% RSLogix 500 project EDINBURG.RSS, saved by version 10.00.00.00 %
PROJECT "EDINBURG"    % processor: MicroLogix 1400 %

PROGRAM FILES
  LAD 2 "MAIN"  12 rungs
  LAD 3 "START/MODE"  11 rungs
  LAD 4 "ENCODER"  11 rungs
  LAD 5 "CRADLE"  25 rungs
  LAD 6 "BRUSH"  8 rungs
  LAD 7 "TANK"  17 rungs
  LAD 8 "AUXILARY"  4 rungs
  LAD 9 "FAULTS"  35 rungs
  LAD 10 "SPARE"  2 rungs
  LAD 11 "DECLINE"  49 rungs
  LAD 12 "STACK LS"  13 rungs
  LAD 13 "STACK"  23 rungs

DATA FILES
  O0 OUTPUT  9 elements
  I1 INPUT  11 elements
  S2 STATUS  66 elements
  B3 BINARY  7 elements
  T4 TIMER  38 elements
  C5 COUNTER  1 elements
  R6 CONTROL  1 elements
  N7 INTEGER  40 elements
  F8 FLOAT  30 elements
  L9   1 elements
  L10   2 elements

LADDER 2 "MAIN"
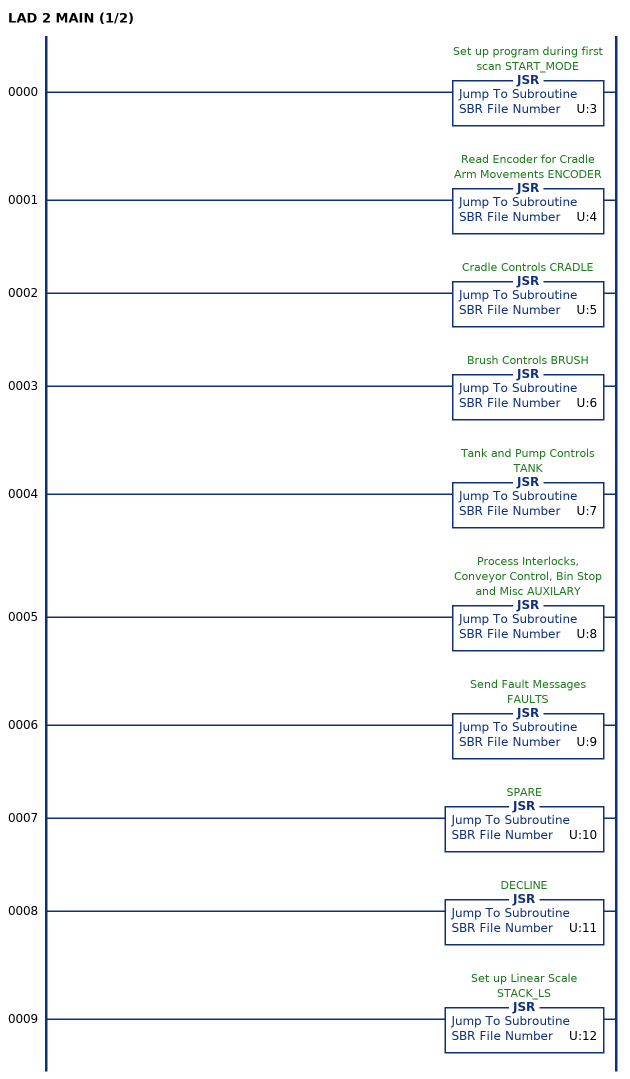
% Rung: 0 %
SOR JSR U:3 EOR
%   U:3  START_MODE  "Set up program during first scan" %
% Rung: 1 %
SOR JSR U:4 EOR
%   U:4  ENCODER  "Read Encoder for Cradle Arm Movements" %
% Rung: 2 %
SOR JSR U:5 EOR
%   U:5  CRADLE  "Cradle Controls" %
% Rung: 3 %
SOR JSR U:6 EOR
%   U:6  BRUSH  "Brush Controls" %
% Rung: 4 %
SOR JSR U:7 EOR
%   U:7  TANK  "Tank and Pump Controls" %
% Rung: 5 %
SOR JSR U:8 EOR
%   U:8  AUXILARY  "Process Interlocks, Conveyor Control, Bin Stop and Misc" %
% Rung: 6 %
SOR JSR U:9 EOR
%   U:9  FAULTS  "Send Fault Messages" %
% Rung: 7 %
SOR JSR U:10 EOR
%   U:10  SPARE %
% Rung: 8 %
SOR JSR U:11 EOR
%   U:11  DECLINE %
% Rung: 9 %
SOR JSR U:12 EOR
%   U:12  STACK_LS  "Set up Linear Scale" %

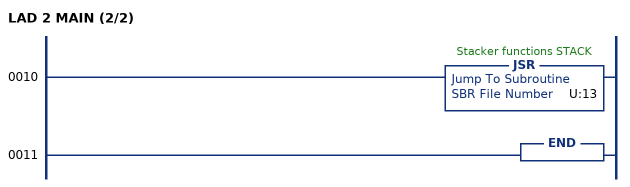
% Rung: 10 %
SOR JSR U:13 EOR
%   U:13  STACK  "Stacker functions" %
% Rung: 11 %
SOR END EOR

LADDER 3 "START/MODE"
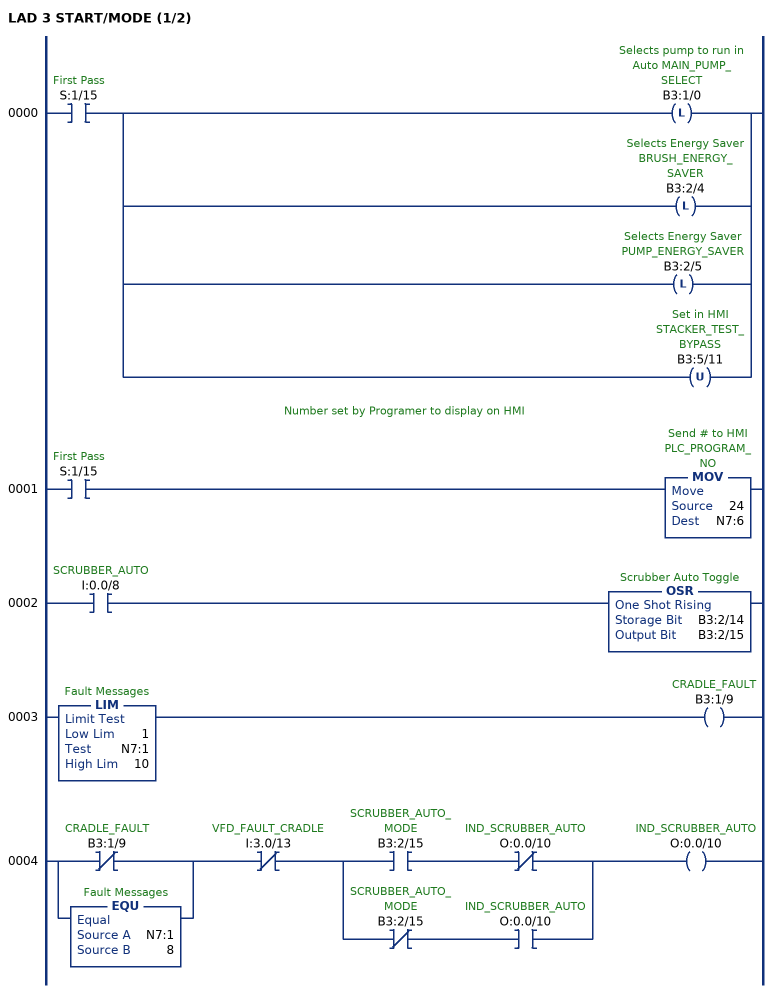
% Rung: 0 %
SOR XIC S:1/15 BST OTL B3:1/0 NXB BST OTL B3:2/4 NXB BST OTL B3:2/5 NXB OTU B3:5/11 BND BND BND EOR
%   S:1/15  "First Pass" %
%   B3:1/0  MAIN_PUMP_SELECT  "Selects pump to run in Auto" %
%   B3:2/4  BRUSH_ENERGY_SAVER  "Selects Energy Saver" %
%   B3:2/5  PUMP_ENERGY_SAVER  "Selects Energy Saver" %
%   B3:5/11  STACKER_TEST_BYPASS  "Set in HMI" %
% Rung: 1 %
% Number set by Programer to display on HMI %
SOR XIC S:1/15 MOV 24 N7:6 EOR
%   S:1/15  "First Pass" %
%   N7:6  PLC_PROGRAM_NO  "Send # to HMI" %
% Rung: 2 %
SOR XIC I:0.0/8 OSR B3:2/14 B3:2/15 EOR
%   I:0.0/8  SCRUBBER_AUTO %
%   B3:2/14  "Scrubber Auto Toggle" %
%   B3:2/15  SCRUBBER_AUTO_MODE %
% Rung: 3 %
SOR LIM 1 N7:1 10 OTE B3:1/9 EOR
%   N7:1  "Fault Messages" %
%   B3:1/9  CRADLE_FAULT %
% Rung: 4 %
SOR BST XIO B3:1/9 NXB EQU N7:1 8 BND XIO I:3.0/13 BST XIC B3:2/15 XIO O:0.0/10 NXB XIO B3:2/15 XIC O:0.0/10 BND OTE O:0.0/10 EOR
%   B3:1/9  CRADLE_FAULT %
%   N7:1  "Fault Messages" %
%   I:3.0/13  VFD_FAULT_CRADLE %
%   B3:2/15  SCRUBBER_AUTO_MODE %
%   O:0.0/10  IND_SCRUBBER_AUTO %

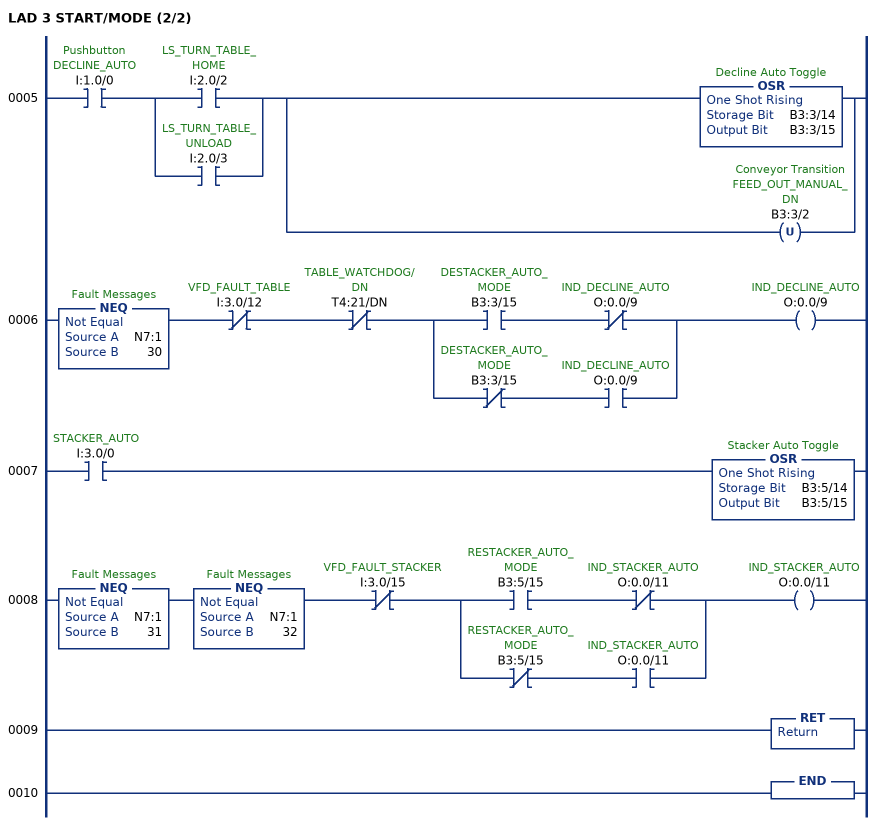
% Rung: 5 %
SOR XIC I:1.0/0 BST XIC I:2.0/2 NXB XIC I:2.0/3 BND BST OSR B3:3/14 B3:3/15 NXB OTU B3:3/2 BND EOR
%   I:1.0/0  DECLINE_AUTO  "Pushbutton" %
%   I:2.0/2  LS_TURN_TABLE_HOME %
%   I:2.0/3  LS_TURN_TABLE_UNLOAD %
%   B3:3/14  "Decline Auto Toggle" %
%   B3:3/15  DESTACKER_AUTO_MODE %
%   B3:3/2  FEED_OUT_MANUAL_DN  "Conveyor Transition" %
% Rung: 6 %
SOR NEQ N7:1 30 XIO I:3.0/12 XIO T4:21/DN BST XIC B3:3/15 XIO O:0.0/9 NXB XIO B3:3/15 XIC O:0.0/9 BND OTE O:0.0/9 EOR
%   N7:1  "Fault Messages" %
%   I:3.0/12  VFD_FAULT_TABLE %
%   T4:21  TABLE_WATCHDOG %
%   B3:3/15  DESTACKER_AUTO_MODE %
%   O:0.0/9  IND_DECLINE_AUTO %
% Rung: 7 %
SOR XIC I:3.0/0 OSR B3:5/14 B3:5/15 EOR
%   I:3.0/0  STACKER_AUTO %
%   B3:5/14  "Stacker Auto Toggle" %
%   B3:5/15  RESTACKER_AUTO_MODE %
% Rung: 8 %
SOR NEQ N7:1 31 NEQ N7:1 32 XIO I:3.0/15 BST XIC B3:5/15 XIO O:0.0/11 NXB XIO B3:5/15 XIC O:0.0/11 BND OTE O:0.0/11 EOR
%   N7:1  "Fault Messages" %
%   I:3.0/15  VFD_FAULT_STACKER %
%   B3:5/15  RESTACKER_AUTO_MODE %
%   O:0.0/11  IND_STACKER_AUTO %
% Rung: 9 %
SOR RET EOR
% Rung: 10 %
SOR END EOR

LADDER 4 "ENCODER"
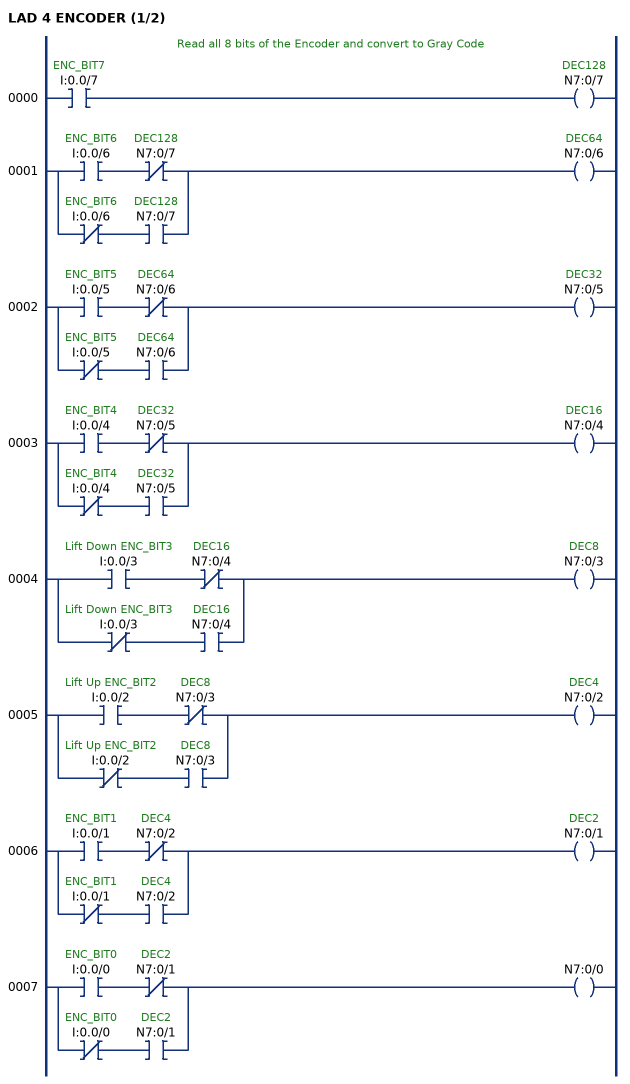
% Rung: 0 %
% Read all 8 bits of the Encoder and convert to Gray Code %
SOR XIC I:0.0/7 OTE N7:0/7 EOR
%   I:0.0/7  ENC_BIT7 %
%   N7:0/7  "DEC128" %
% Rung: 1 %
SOR BST XIC I:0.0/6 XIO N7:0/7 NXB XIO I:0.0/6 XIC N7:0/7 BND OTE N7:0/6 EOR
%   I:0.0/6  ENC_BIT6 %
%   N7:0/7  "DEC128" %
%   N7:0/6  "DEC64" %
% Rung: 2 %
SOR BST XIC I:0.0/5 XIO N7:0/6 NXB XIO I:0.0/5 XIC N7:0/6 BND OTE N7:0/5 EOR
%   I:0.0/5  ENC_BIT5 %
%   N7:0/6  "DEC64" %
%   N7:0/5  "DEC32" %
% Rung: 3 %
SOR BST XIC I:0.0/4 XIO N7:0/5 NXB XIO I:0.0/4 XIC N7:0/5 BND OTE N7:0/4 EOR
%   I:0.0/4  ENC_BIT4 %
%   N7:0/5  "DEC32" %
%   N7:0/4  "DEC16" %
% Rung: 4 %
SOR BST XIC I:0.0/3 XIO N7:0/4 NXB XIO I:0.0/3 XIC N7:0/4 BND OTE N7:0/3 EOR
%   I:0.0/3  ENC_BIT3  "Lift Down" %
%   N7:0/4  "DEC16" %
%   N7:0/3  "DEC8" %
% Rung: 5 %
SOR BST XIC I:0.0/2 XIO N7:0/3 NXB XIO I:0.0/2 XIC N7:0/3 BND OTE N7:0/2 EOR
%   I:0.0/2  ENC_BIT2  "Lift Up" %
%   N7:0/3  "DEC8" %
%   N7:0/2  "DEC4" %
% Rung: 6 %
SOR BST XIC I:0.0/1 XIO N7:0/2 NXB XIO I:0.0/1 XIC N7:0/2 BND OTE N7:0/1 EOR
%   I:0.0/1  ENC_BIT1 %
%   N7:0/2  "DEC4" %
%   N7:0/1  "DEC2" %
% Rung: 7 %
SOR BST XIC I:0.0/0 XIO N7:0/1 NXB XIO I:0.0/0 XIC N7:0/1 BND OTE N7:0/0 EOR
%   I:0.0/0  ENC_BIT0 %
%   N7:0/1  "DEC2" %

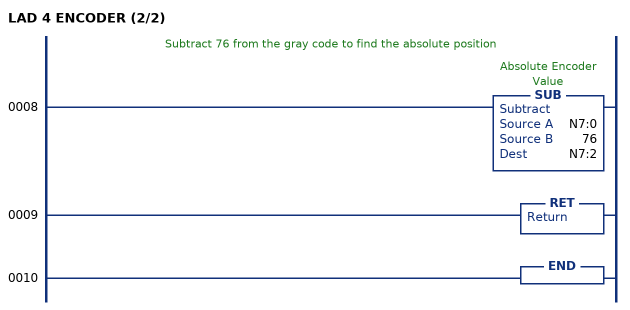
% Rung: 8 %
% Subtract 76 from the gray code to find the absolute position %
SOR SUB N7:0 76 N7:2 EOR
%   N7:0  ENC_POS %
%   N7:2  "Absolute Encoder Value" %
% Rung: 9 %
SOR RET EOR
% Rung: 10 %
SOR END EOR

LADDER 5 "CRADLE"
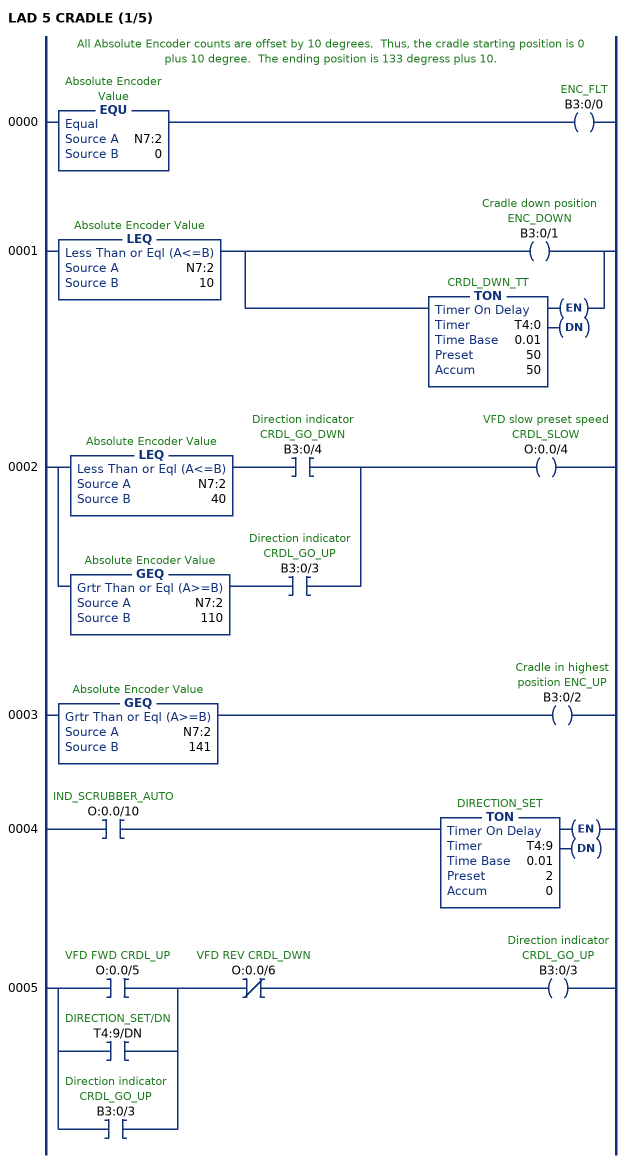
% Rung: 0 %
% All Absolute Encoder counts are offset by 10 degrees.  Thus, the cradle starting position is 0 plus 10 degree.  The ending position is 133 degress plus 10. %
SOR EQU N7:2 0 OTE B3:0/0 EOR
%   N7:2  "Absolute Encoder Value" %
%   B3:0/0  ENC_FLT %
% Rung: 1 %
SOR LEQ N7:2 10 BST OTE B3:0/1 NXB TON T4:0 0.01 50 50 BND EOR
%   N7:2  "Absolute Encoder Value" %
%   B3:0/1  ENC_DOWN  "Cradle down position" %
%   T4:0  CRDL_DWN_TT %
% Rung: 2 %
SOR BST LEQ N7:2 40 XIC B3:0/4 NXB GEQ N7:2 110 XIC B3:0/3 BND OTE O:0.0/4 EOR
%   N7:2  "Absolute Encoder Value" %
%   B3:0/4  CRDL_GO_DWN  "Direction indicator" %
%   B3:0/3  CRDL_GO_UP  "Direction indicator" %
%   O:0.0/4  CRDL_SLOW  "VFD slow preset speed" %
% Rung: 3 %
SOR GEQ N7:2 141 OTE B3:0/2 EOR
%   N7:2  "Absolute Encoder Value" %
%   B3:0/2  ENC_UP  "Cradle in highest position" %
% Rung: 4 %
SOR XIC O:0.0/10 TON T4:9 0.01 2 0 EOR
%   O:0.0/10  IND_SCRUBBER_AUTO %
%   T4:9  DIRECTION_SET %
% Rung: 5 %
SOR BST XIC O:0.0/5 NXB XIC T4:9/DN NXB XIC B3:0/3 BND XIO O:0.0/6 OTE B3:0/3 EOR
%   O:0.0/5  CRDL_UP  "VFD FWD" %
%   T4:9  DIRECTION_SET %
%   B3:0/3  CRDL_GO_UP  "Direction indicator" %
%   O:0.0/6  CRDL_DWN  "VFD REV" %

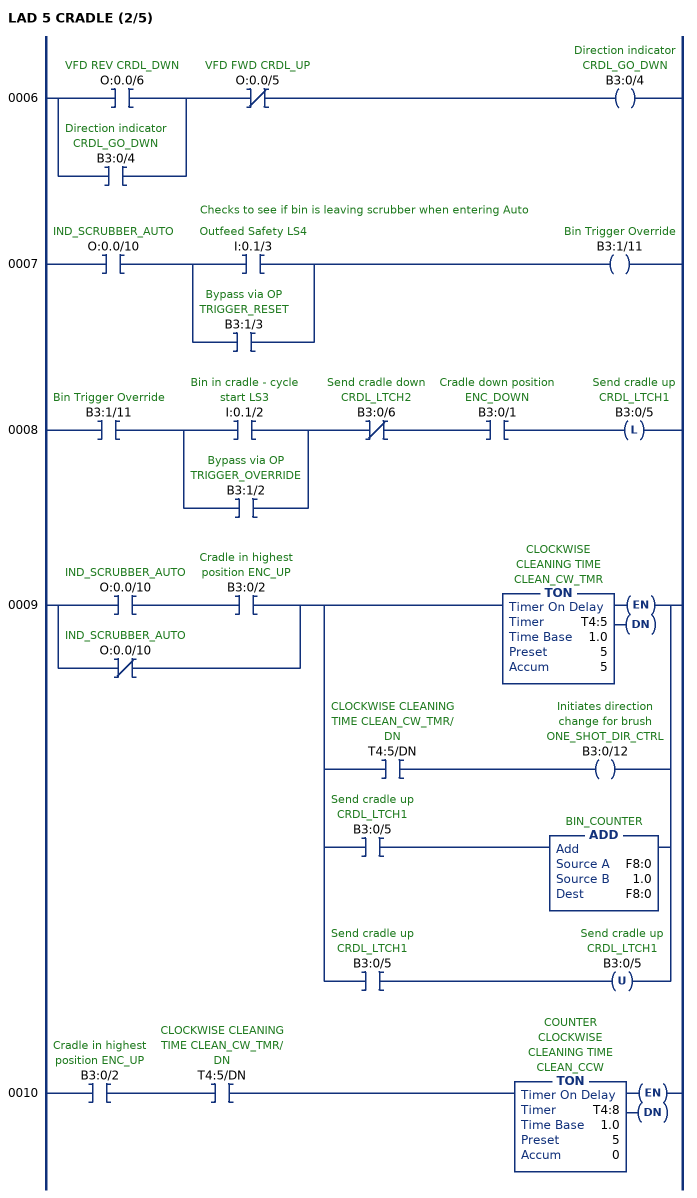
% Rung: 6 %
SOR BST XIC O:0.0/6 NXB XIC B3:0/4 BND XIO O:0.0/5 OTE B3:0/4 EOR
%   O:0.0/6  CRDL_DWN  "VFD REV" %
%   B3:0/4  CRDL_GO_DWN  "Direction indicator" %
%   O:0.0/5  CRDL_UP  "VFD FWD" %
% Rung: 7 %
% Checks to see if bin is leaving scrubber when entering Auto %
SOR XIC O:0.0/10 BST XIC I:0.1/3 NXB XIC B3:1/3 BND OTE B3:1/11 EOR
%   O:0.0/10  IND_SCRUBBER_AUTO %
%   I:0.1/3  LS4  "Outfeed Safety" %
%   B3:1/3  TRIGGER_RESET  "Bypass via OP" %
%   B3:1/11  "Bin Trigger Override" %
% Rung: 8 %
SOR XIC B3:1/11 BST XIC I:0.1/2 NXB XIC B3:1/2 BND XIO B3:0/6 XIC B3:0/1 OTL B3:0/5 EOR
%   B3:1/11  "Bin Trigger Override" %
%   I:0.1/2  LS3  "Bin in cradle - cycle start" %
%   B3:1/2  TRIGGER_OVERRIDE  "Bypass via OP" %
%   B3:0/6  CRDL_LTCH2  "Send cradle down" %
%   B3:0/1  ENC_DOWN  "Cradle down position" %
%   B3:0/5  CRDL_LTCH1  "Send cradle up" %
% Rung: 9 %
SOR BST XIC O:0.0/10 XIC B3:0/2 NXB XIO O:0.0/10 BND BST TON T4:5 1.0 5 5 NXB XIC T4:5/DN OTE B3:0/12 NXB BST XIC B3:0/5 ADD F8:0 1.0 F8:0 NXB XIC B3:0/5 OTU B3:0/5 BND BND EOR
%   O:0.0/10  IND_SCRUBBER_AUTO %
%   B3:0/2  ENC_UP  "Cradle in highest position" %
%   T4:5  CLEAN_CW_TMR  "CLOCKWISE CLEANING TIME" %
%   B3:0/12  ONE_SHOT_DIR_CTRL  "Initiates direction change for brush" %
%   B3:0/5  CRDL_LTCH1  "Send cradle up" %
%   F8:0  BIN_COUNTER %
% Rung: 10 %
SOR XIC B3:0/2 XIC T4:5/DN TON T4:8 1.0 5 0 EOR
%   B3:0/2  ENC_UP  "Cradle in highest position" %
%   T4:5  CLEAN_CW_TMR  "CLOCKWISE CLEANING TIME" %
%   T4:8  CLEAN_CCW  "COUNTER CLOCKWISE CLEANING TIME" %

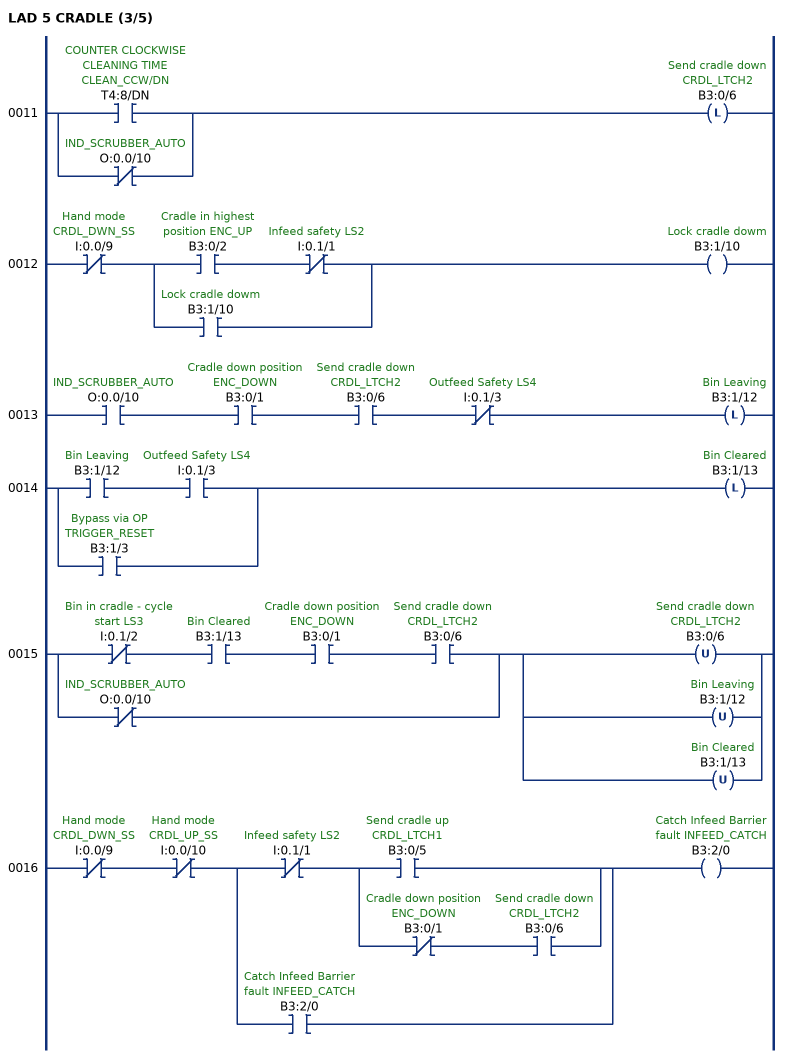
% Rung: 11 %
SOR BST XIC T4:8/DN NXB XIO O:0.0/10 BND OTL B3:0/6 EOR
%   T4:8  CLEAN_CCW  "COUNTER CLOCKWISE CLEANING TIME" %
%   O:0.0/10  IND_SCRUBBER_AUTO %
%   B3:0/6  CRDL_LTCH2  "Send cradle down" %
% Rung: 12 %
SOR XIO I:0.0/9 BST XIC B3:0/2 XIO I:0.1/1 NXB XIC B3:1/10 BND OTE B3:1/10 EOR
%   I:0.0/9  CRDL_DWN_SS  "Hand mode" %
%   B3:0/2  ENC_UP  "Cradle in highest position" %
%   I:0.1/1  LS2  "Infeed safety" %
%   B3:1/10  "Lock cradle dowm" %
% Rung: 13 %
SOR XIC O:0.0/10 XIC B3:0/1 XIC B3:0/6 XIO I:0.1/3 OTL B3:1/12 EOR
%   O:0.0/10  IND_SCRUBBER_AUTO %
%   B3:0/1  ENC_DOWN  "Cradle down position" %
%   B3:0/6  CRDL_LTCH2  "Send cradle down" %
%   I:0.1/3  LS4  "Outfeed Safety" %
%   B3:1/12  "Bin Leaving" %
% Rung: 14 %
SOR BST XIC B3:1/12 XIC I:0.1/3 NXB XIC B3:1/3 BND OTL B3:1/13 EOR
%   B3:1/12  "Bin Leaving" %
%   I:0.1/3  LS4  "Outfeed Safety" %
%   B3:1/3  TRIGGER_RESET  "Bypass via OP" %
%   B3:1/13  "Bin Cleared" %
% Rung: 15 %
SOR BST XIO I:0.1/2 XIC B3:1/13 XIC B3:0/1 XIC B3:0/6 NXB XIO O:0.0/10 BND BST OTU B3:0/6 NXB BST OTU B3:1/12 NXB OTU B3:1/13 BND BND EOR
%   I:0.1/2  LS3  "Bin in cradle - cycle start" %
%   B3:1/13  "Bin Cleared" %
%   B3:0/1  ENC_DOWN  "Cradle down position" %
%   B3:0/6  CRDL_LTCH2  "Send cradle down" %
%   O:0.0/10  IND_SCRUBBER_AUTO %
%   B3:1/12  "Bin Leaving" %
% Rung: 16 %
SOR XIO I:0.0/9 XIO I:0.0/10 BST XIO I:0.1/1 BST XIC B3:0/5 NXB XIO B3:0/1 XIC B3:0/6 BND NXB XIC B3:2/0 BND OTE B3:2/0 EOR
%   I:0.0/9  CRDL_DWN_SS  "Hand mode" %
%   I:0.0/10  CRDL_UP_SS  "Hand mode" %
%   I:0.1/1  LS2  "Infeed safety" %
%   B3:0/5  CRDL_LTCH1  "Send cradle up" %
%   B3:0/1  ENC_DOWN  "Cradle down position" %
%   B3:0/6  CRDL_LTCH2  "Send cradle down" %
%   B3:2/0  INFEED_CATCH  "Catch Infeed Barrier fault" %

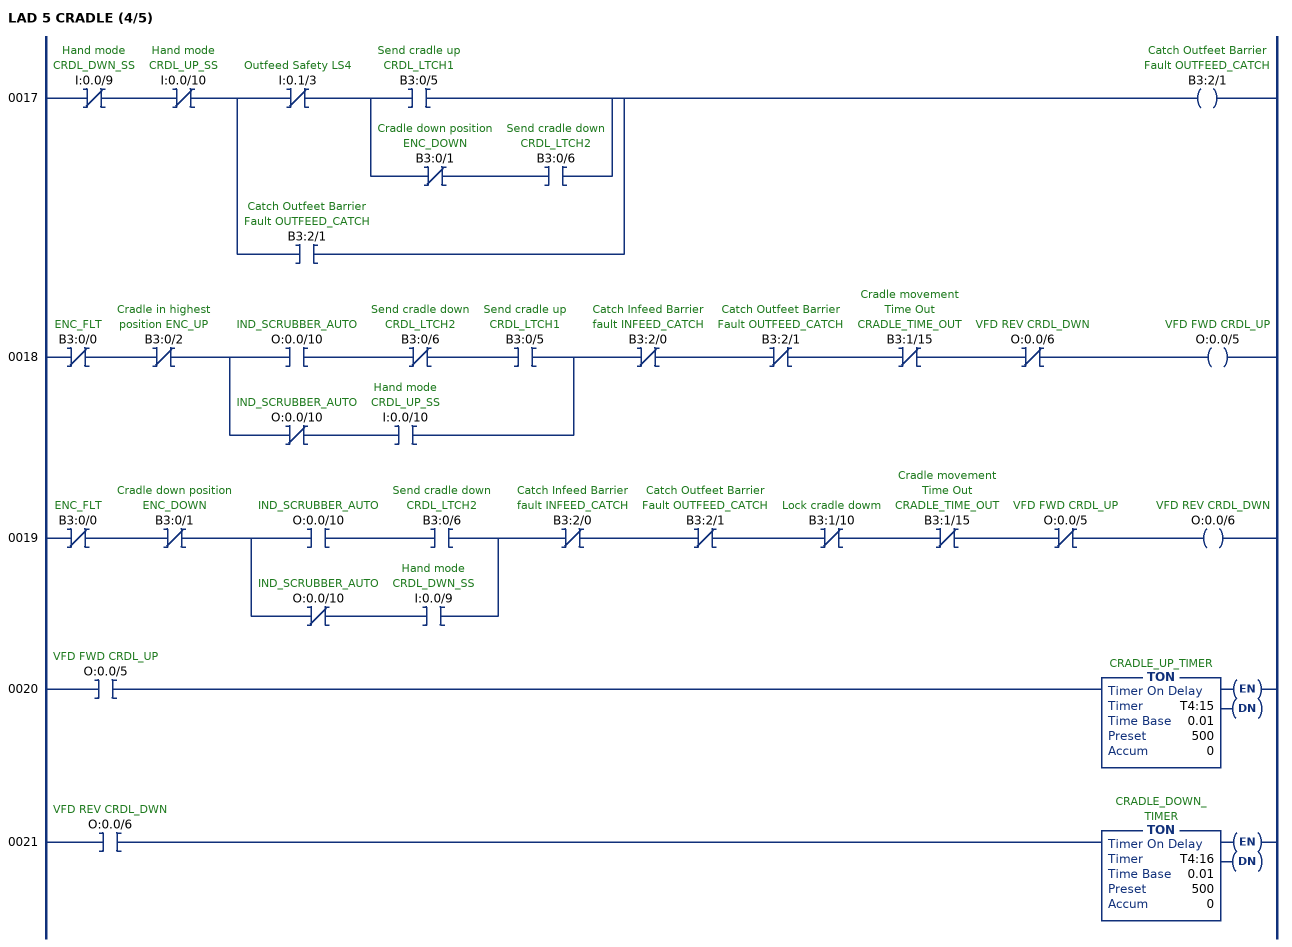
% Rung: 17 %
SOR XIO I:0.0/9 XIO I:0.0/10 BST XIO I:0.1/3 BST XIC B3:0/5 NXB XIO B3:0/1 XIC B3:0/6 BND NXB XIC B3:2/1 BND OTE B3:2/1 EOR
%   I:0.0/9  CRDL_DWN_SS  "Hand mode" %
%   I:0.0/10  CRDL_UP_SS  "Hand mode" %
%   I:0.1/3  LS4  "Outfeed Safety" %
%   B3:0/5  CRDL_LTCH1  "Send cradle up" %
%   B3:0/1  ENC_DOWN  "Cradle down position" %
%   B3:0/6  CRDL_LTCH2  "Send cradle down" %
%   B3:2/1  OUTFEED_CATCH  "Catch Outfeet Barrier Fault" %
% Rung: 18 %
SOR XIO B3:0/0 XIO B3:0/2 BST XIC O:0.0/10 XIO B3:0/6 XIC B3:0/5 NXB XIO O:0.0/10 XIC I:0.0/10 BND XIO B3:2/0 XIO B3:2/1 XIO B3:1/15 XIO O:0.0/6 OTE O:0.0/5 EOR
%   B3:0/0  ENC_FLT %
%   B3:0/2  ENC_UP  "Cradle in highest position" %
%   O:0.0/10  IND_SCRUBBER_AUTO %
%   B3:0/6  CRDL_LTCH2  "Send cradle down" %
%   B3:0/5  CRDL_LTCH1  "Send cradle up" %
%   I:0.0/10  CRDL_UP_SS  "Hand mode" %
%   B3:2/0  INFEED_CATCH  "Catch Infeed Barrier fault" %
%   B3:2/1  OUTFEED_CATCH  "Catch Outfeet Barrier Fault" %
%   B3:1/15  CRADLE_TIME_OUT  "Cradle movement Time Out" %
%   O:0.0/6  CRDL_DWN  "VFD REV" %
%   O:0.0/5  CRDL_UP  "VFD FWD" %
% Rung: 19 %
SOR XIO B3:0/0 XIO B3:0/1 BST XIC O:0.0/10 XIC B3:0/6 NXB XIO O:0.0/10 XIC I:0.0/9 BND XIO B3:2/0 XIO B3:2/1 XIO B3:1/10 XIO B3:1/15 XIO O:0.0/5 OTE O:0.0/6 EOR
%   B3:0/0  ENC_FLT %
%   B3:0/1  ENC_DOWN  "Cradle down position" %
%   O:0.0/10  IND_SCRUBBER_AUTO %
%   B3:0/6  CRDL_LTCH2  "Send cradle down" %
%   I:0.0/9  CRDL_DWN_SS  "Hand mode" %
%   B3:2/0  INFEED_CATCH  "Catch Infeed Barrier fault" %
%   B3:2/1  OUTFEED_CATCH  "Catch Outfeet Barrier Fault" %
%   B3:1/10  "Lock cradle dowm" %
%   B3:1/15  CRADLE_TIME_OUT  "Cradle movement Time Out" %
%   O:0.0/5  CRDL_UP  "VFD FWD" %
%   O:0.0/6  CRDL_DWN  "VFD REV" %
% Rung: 20 %
SOR XIC O:0.0/5 TON T4:15 0.01 500 0 EOR
%   O:0.0/5  CRDL_UP  "VFD FWD" %
%   T4:15  CRADLE_UP_TIMER %
% Rung: 21 %
SOR XIC O:0.0/6 TON T4:16 0.01 500 0 EOR
%   O:0.0/6  CRDL_DWN  "VFD REV" %
%   T4:16  CRADLE_DOWN_TIMER %

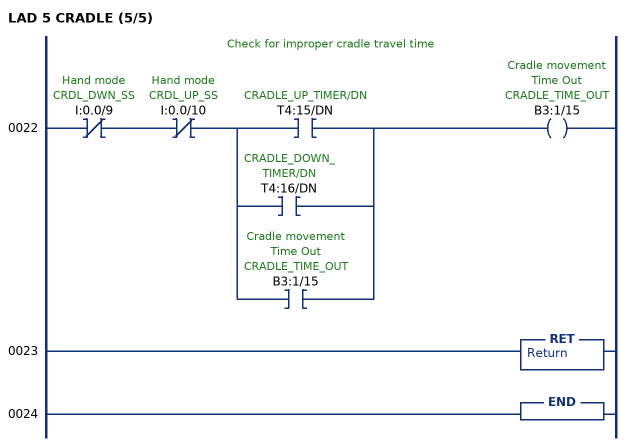
% Rung: 22 %
% Check for improper cradle travel time %
SOR XIO I:0.0/9 XIO I:0.0/10 BST BST XIC T4:15/DN NXB XIC T4:16/DN BND NXB XIC B3:1/15 BND OTE B3:1/15 EOR
%   I:0.0/9  CRDL_DWN_SS  "Hand mode" %
%   I:0.0/10  CRDL_UP_SS  "Hand mode" %
%   T4:15  CRADLE_UP_TIMER %
%   T4:16  CRADLE_DOWN_TIMER %
%   B3:1/15  CRADLE_TIME_OUT  "Cradle movement Time Out" %
% Rung: 23 %
SOR RET EOR
% Rung: 24 %
SOR END EOR

LADDER 6 "BRUSH"
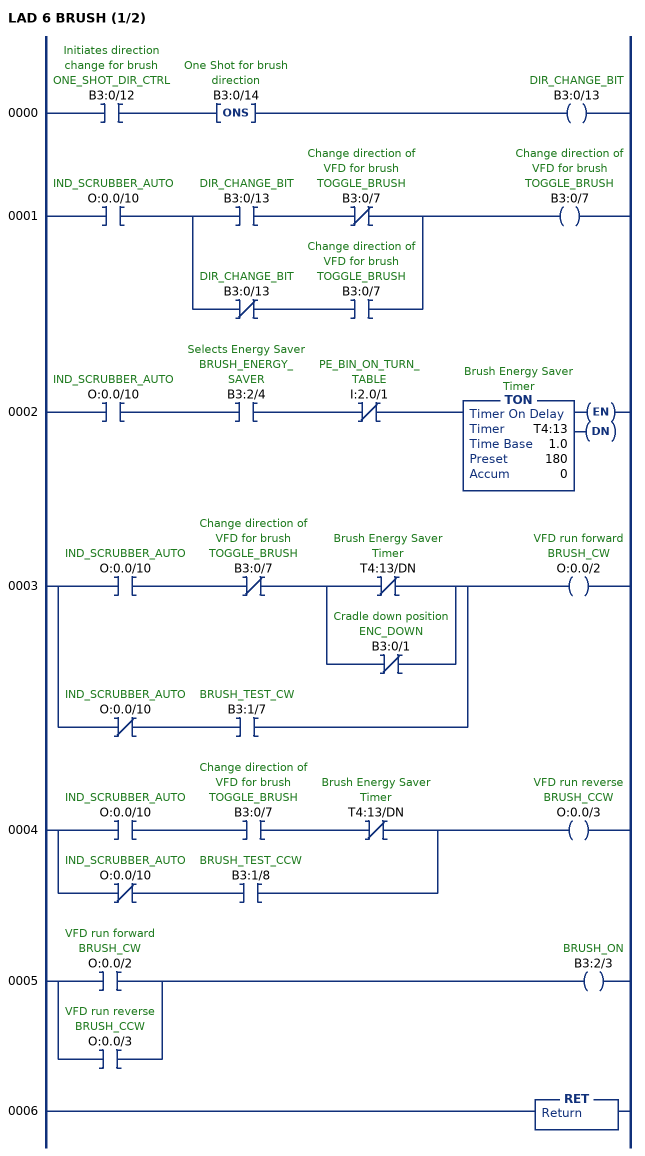
% Rung: 0 %
SOR XIC B3:0/12 ONS B3:0/14 OTE B3:0/13 EOR
%   B3:0/12  ONE_SHOT_DIR_CTRL  "Initiates direction change for brush" %
%   B3:0/14  "One Shot for brush direction" %
%   B3:0/13  DIR_CHANGE_BIT %
% Rung: 1 %
SOR XIC O:0.0/10 BST XIC B3:0/13 XIO B3:0/7 NXB XIO B3:0/13 XIC B3:0/7 BND OTE B3:0/7 EOR
%   O:0.0/10  IND_SCRUBBER_AUTO %
%   B3:0/13  DIR_CHANGE_BIT %
%   B3:0/7  TOGGLE_BRUSH  "Change direction of VFD for brush" %
% Rung: 2 %
SOR XIC O:0.0/10 XIC B3:2/4 XIO I:2.0/1 TON T4:13 1.0 180 0 EOR
%   O:0.0/10  IND_SCRUBBER_AUTO %
%   B3:2/4  BRUSH_ENERGY_SAVER  "Selects Energy Saver" %
%   I:2.0/1  PE_BIN_ON_TURN_TABLE %
%   T4:13  "Brush Energy Saver Timer" %
% Rung: 3 %
SOR BST XIC O:0.0/10 XIO B3:0/7 BST XIO T4:13/DN NXB XIO B3:0/1 BND NXB XIO O:0.0/10 XIC B3:1/7 BND OTE O:0.0/2 EOR
%   O:0.0/10  IND_SCRUBBER_AUTO %
%   B3:0/7  TOGGLE_BRUSH  "Change direction of VFD for brush" %
%   T4:13  "Brush Energy Saver Timer" %
%   B3:0/1  ENC_DOWN  "Cradle down position" %
%   B3:1/7  BRUSH_TEST_CW %
%   O:0.0/2  BRUSH_CW  "VFD run forward" %
% Rung: 4 %
SOR BST XIC O:0.0/10 XIC B3:0/7 XIO T4:13/DN NXB XIO O:0.0/10 XIC B3:1/8 BND OTE O:0.0/3 EOR
%   O:0.0/10  IND_SCRUBBER_AUTO %
%   B3:0/7  TOGGLE_BRUSH  "Change direction of VFD for brush" %
%   T4:13  "Brush Energy Saver Timer" %
%   B3:1/8  BRUSH_TEST_CCW %
%   O:0.0/3  BRUSH_CCW  "VFD run reverse" %
% Rung: 5 %
SOR BST XIC O:0.0/2 NXB XIC O:0.0/3 BND OTE B3:2/3 EOR
%   O:0.0/2  BRUSH_CW  "VFD run forward" %
%   O:0.0/3  BRUSH_CCW  "VFD run reverse" %
%   B3:2/3  BRUSH_ON %
% Rung: 6 %
SOR RET EOR

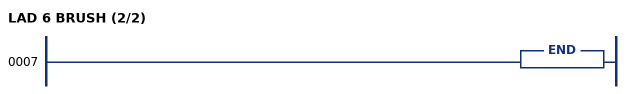
% Rung: 7 %
SOR END EOR

LADDER 7 "TANK"
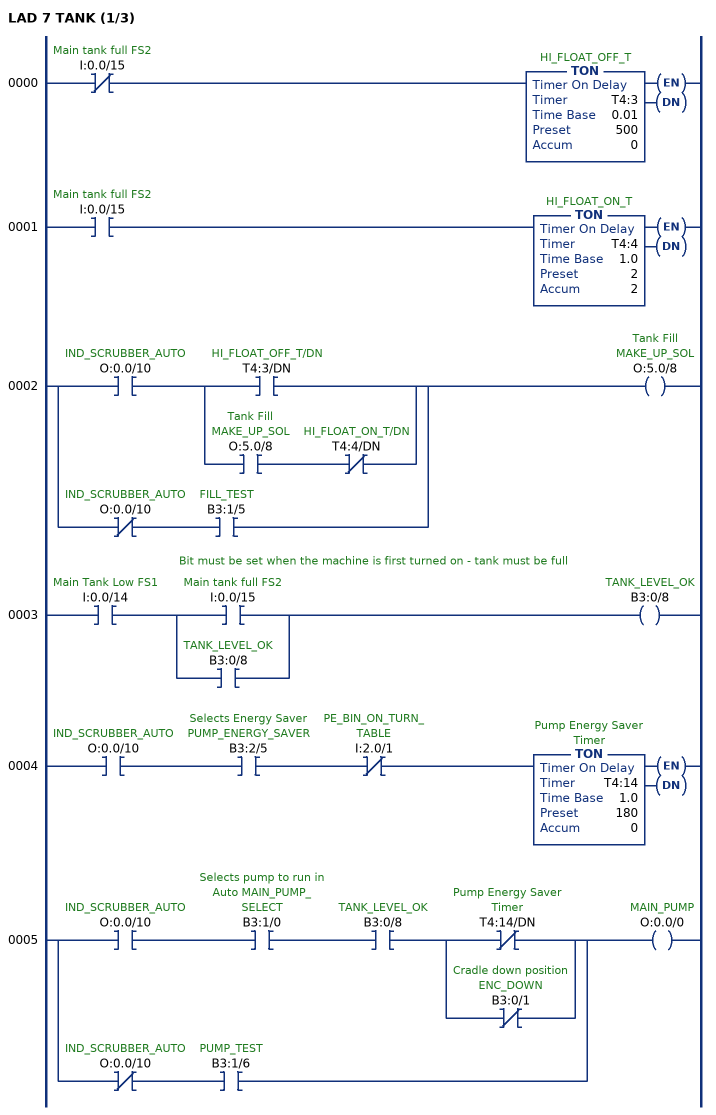
% Rung: 0 %
SOR XIO I:0.0/15 TON T4:3 0.01 500 0 EOR
%   I:0.0/15  FS2  "Main tank full" %
%   T4:3  HI_FLOAT_OFF_T %
% Rung: 1 %
SOR XIC I:0.0/15 TON T4:4 1.0 2 2 EOR
%   I:0.0/15  FS2  "Main tank full" %
%   T4:4  HI_FLOAT_ON_T %
% Rung: 2 %
SOR BST XIC O:0.0/10 BST XIC T4:3/DN NXB XIC O:5.0/8 XIO T4:4/DN BND NXB XIO O:0.0/10 XIC B3:1/5 BND OTE O:5.0/8 EOR
%   O:0.0/10  IND_SCRUBBER_AUTO %
%   T4:3  HI_FLOAT_OFF_T %
%   O:5.0/8  MAKE_UP_SOL  "Tank Fill" %
%   T4:4  HI_FLOAT_ON_T %
%   B3:1/5  FILL_TEST %
% Rung: 3 %
% Bit must be set when the machine is first turned on - tank must be full %
SOR XIC I:0.0/14 BST XIC I:0.0/15 NXB XIC B3:0/8 BND OTE B3:0/8 EOR
%   I:0.0/14  FS1  "Main Tank Low" %
%   I:0.0/15  FS2  "Main tank full" %
%   B3:0/8  TANK_LEVEL_OK %
% Rung: 4 %
SOR XIC O:0.0/10 XIC B3:2/5 XIO I:2.0/1 TON T4:14 1.0 180 0 EOR
%   O:0.0/10  IND_SCRUBBER_AUTO %
%   B3:2/5  PUMP_ENERGY_SAVER  "Selects Energy Saver" %
%   I:2.0/1  PE_BIN_ON_TURN_TABLE %
%   T4:14  "Pump Energy Saver Timer" %
% Rung: 5 %
SOR BST XIC O:0.0/10 XIC B3:1/0 XIC B3:0/8 BST XIO T4:14/DN NXB XIO B3:0/1 BND NXB XIO O:0.0/10 XIC B3:1/6 BND OTE O:0.0/0 EOR
%   O:0.0/10  IND_SCRUBBER_AUTO %
%   B3:1/0  MAIN_PUMP_SELECT  "Selects pump to run in Auto" %
%   B3:0/8  TANK_LEVEL_OK %
%   T4:14  "Pump Energy Saver Timer" %
%   B3:0/1  ENC_DOWN  "Cradle down position" %
%   B3:1/6  PUMP_TEST %
%   O:0.0/0  MAIN_PUMP %

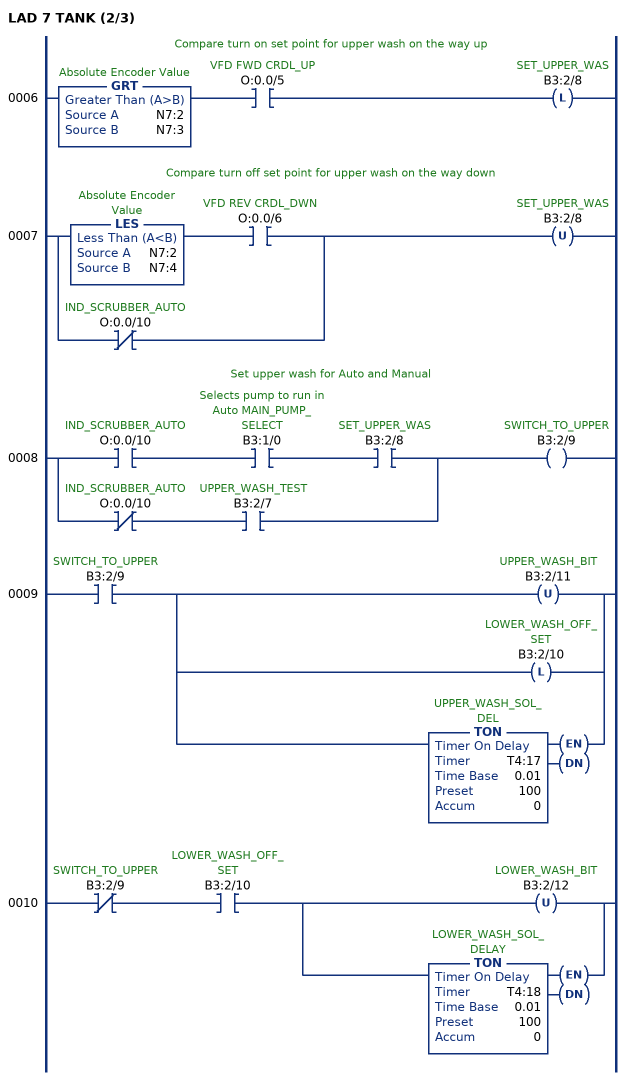
% Rung: 6 %
% Compare turn on set point for upper wash on the way up %
SOR GRT N7:2 N7:3 XIC O:0.0/5 OTL B3:2/8 EOR
%   N7:2  "Absolute Encoder Value" %
%   N7:3  UPPER_WASH_TURN_ON %
%   O:0.0/5  CRDL_UP  "VFD FWD" %
%   B3:2/8  SET_UPPER_WAS %
% Rung: 7 %
% Compare turn off set point for upper wash on the way down %
SOR BST LES N7:2 N7:4 XIC O:0.0/6 NXB XIO O:0.0/10 BND OTU B3:2/8 EOR
%   N7:2  "Absolute Encoder Value" %
%   N7:4  UPPER_WASH_TURN_OFF %
%   O:0.0/6  CRDL_DWN  "VFD REV" %
%   O:0.0/10  IND_SCRUBBER_AUTO %
%   B3:2/8  SET_UPPER_WAS %
% Rung: 8 %
% Set upper wash for Auto and Manual %
SOR BST XIC O:0.0/10 XIC B3:1/0 XIC B3:2/8 NXB XIO O:0.0/10 XIC B3:2/7 BND OTE B3:2/9 EOR
%   O:0.0/10  IND_SCRUBBER_AUTO %
%   B3:1/0  MAIN_PUMP_SELECT  "Selects pump to run in Auto" %
%   B3:2/8  SET_UPPER_WAS %
%   B3:2/7  UPPER_WASH_TEST %
%   B3:2/9  SWITCH_TO_UPPER %
% Rung: 9 %
SOR XIC B3:2/9 BST OTU B3:2/11 NXB BST OTL B3:2/10 NXB TON T4:17 0.01 100 0 BND BND EOR
%   B3:2/9  SWITCH_TO_UPPER %
%   B3:2/11  UPPER_WASH_BIT %
%   B3:2/10  LOWER_WASH_OFF_SET %
%   T4:17  UPPER_WASH_SOL_DEL %
% Rung: 10 %
SOR XIO B3:2/9 XIC B3:2/10 BST OTU B3:2/12 NXB TON T4:18 0.01 100 0 BND EOR
%   B3:2/9  SWITCH_TO_UPPER %
%   B3:2/10  LOWER_WASH_OFF_SET %
%   B3:2/12  LOWER_WASH_BIT %
%   T4:18  LOWER_WASH_SOL_DELAY %

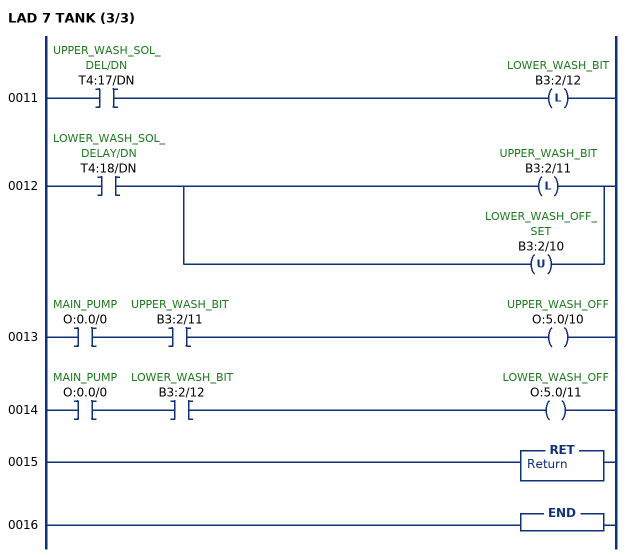
% Rung: 11 %
SOR XIC T4:17/DN OTL B3:2/12 EOR
%   T4:17  UPPER_WASH_SOL_DEL %
%   B3:2/12  LOWER_WASH_BIT %
% Rung: 12 %
SOR XIC T4:18/DN BST OTL B3:2/11 NXB OTU B3:2/10 BND EOR
%   T4:18  LOWER_WASH_SOL_DELAY %
%   B3:2/11  UPPER_WASH_BIT %
%   B3:2/10  LOWER_WASH_OFF_SET %
% Rung: 13 %
SOR XIC O:0.0/0 XIC B3:2/11 OTE O:5.0/10 EOR
%   O:0.0/0  MAIN_PUMP %
%   B3:2/11  UPPER_WASH_BIT %
%   O:5.0/10  UPPER_WASH_OFF %
% Rung: 14 %
SOR XIC O:0.0/0 XIC B3:2/12 OTE O:5.0/11 EOR
%   O:0.0/0  MAIN_PUMP %
%   B3:2/12  LOWER_WASH_BIT %
%   O:5.0/11  LOWER_WASH_OFF %
% Rung: 15 %
SOR RET EOR
% Rung: 16 %
SOR END EOR

LADDER 8 "AUXILARY"
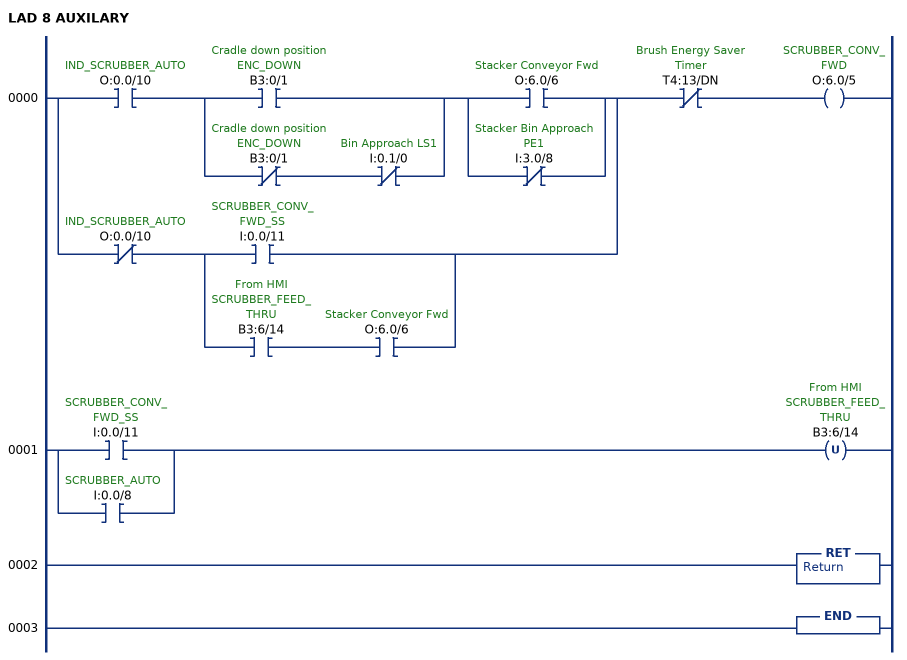
% Rung: 0 %
SOR BST XIC O:0.0/10 BST XIC B3:0/1 NXB XIO B3:0/1 XIO I:0.1/0 BND BST XIC O:6.0/6 NXB XIO I:3.0/8 BND NXB XIO O:0.0/10 BST XIC I:0.0/11 NXB XIC B3:6/14 XIC O:6.0/6 BND BND XIO T4:13/DN OTE O:6.0/5 EOR
%   O:0.0/10  IND_SCRUBBER_AUTO %
%   B3:0/1  ENC_DOWN  "Cradle down position" %
%   I:0.1/0  LS1  "Bin Approach" %
%   O:6.0/6  "Stacker Conveyor Fwd" %
%   I:3.0/8  PE1  "Stacker Bin Approach" %
%   I:0.0/11  SCRUBBER_CONV_FWD_SS %
%   B3:6/14  SCRUBBER_FEED_THRU  "From HMI" %
%   T4:13  "Brush Energy Saver Timer" %
%   O:6.0/5  SCRUBBER_CONV_FWD %
% Rung: 1 %
SOR BST XIC I:0.0/11 NXB XIC I:0.0/8 BND OTU B3:6/14 EOR
%   I:0.0/11  SCRUBBER_CONV_FWD_SS %
%   I:0.0/8  SCRUBBER_AUTO %
%   B3:6/14  SCRUBBER_FEED_THRU  "From HMI" %
% Rung: 2 %
SOR RET EOR
% Rung: 3 %
SOR END EOR

LADDER 9 "FAULTS"
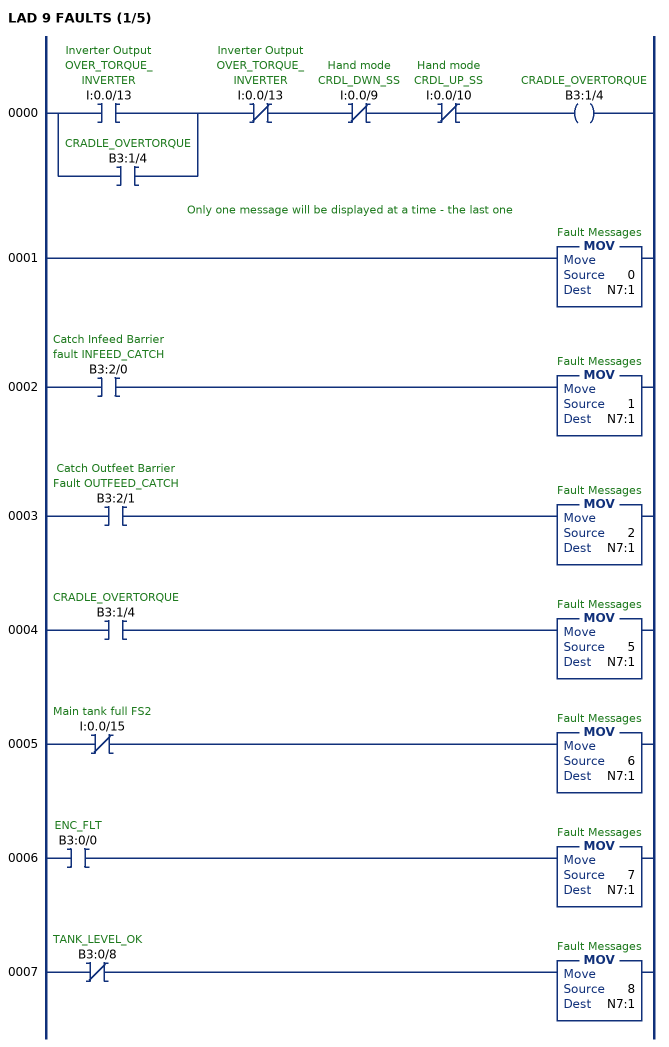
% Rung: 0 %
SOR BST XIC I:0.0/13 NXB XIC B3:1/4 BND XIO I:0.0/13 XIO I:0.0/9 XIO I:0.0/10 OTE B3:1/4 EOR
%   I:0.0/13  OVER_TORQUE_INVERTER  "Inverter Output" %
%   B3:1/4  CRADLE_OVERTORQUE %
%   I:0.0/9  CRDL_DWN_SS  "Hand mode" %
%   I:0.0/10  CRDL_UP_SS  "Hand mode" %
% Rung: 1 %
% Only one message will be displayed at a time - the last one %
SOR MOV 0 N7:1 EOR
%   N7:1  "Fault Messages" %
% Rung: 2 %
SOR XIC B3:2/0 MOV 1 N7:1 EOR
%   B3:2/0  INFEED_CATCH  "Catch Infeed Barrier fault" %
%   N7:1  "Fault Messages" %
% Rung: 3 %
SOR XIC B3:2/1 MOV 2 N7:1 EOR
%   B3:2/1  OUTFEED_CATCH  "Catch Outfeet Barrier Fault" %
%   N7:1  "Fault Messages" %
% Rung: 4 %
SOR XIC B3:1/4 MOV 5 N7:1 EOR
%   B3:1/4  CRADLE_OVERTORQUE %
%   N7:1  "Fault Messages" %
% Rung: 5 %
SOR XIO I:0.0/15 MOV 6 N7:1 EOR
%   I:0.0/15  FS2  "Main tank full" %
%   N7:1  "Fault Messages" %
% Rung: 6 %
SOR XIC B3:0/0 MOV 7 N7:1 EOR
%   B3:0/0  ENC_FLT %
%   N7:1  "Fault Messages" %
% Rung: 7 %
SOR XIO B3:0/8 MOV 8 N7:1 EOR
%   B3:0/8  TANK_LEVEL_OK %
%   N7:1  "Fault Messages" %

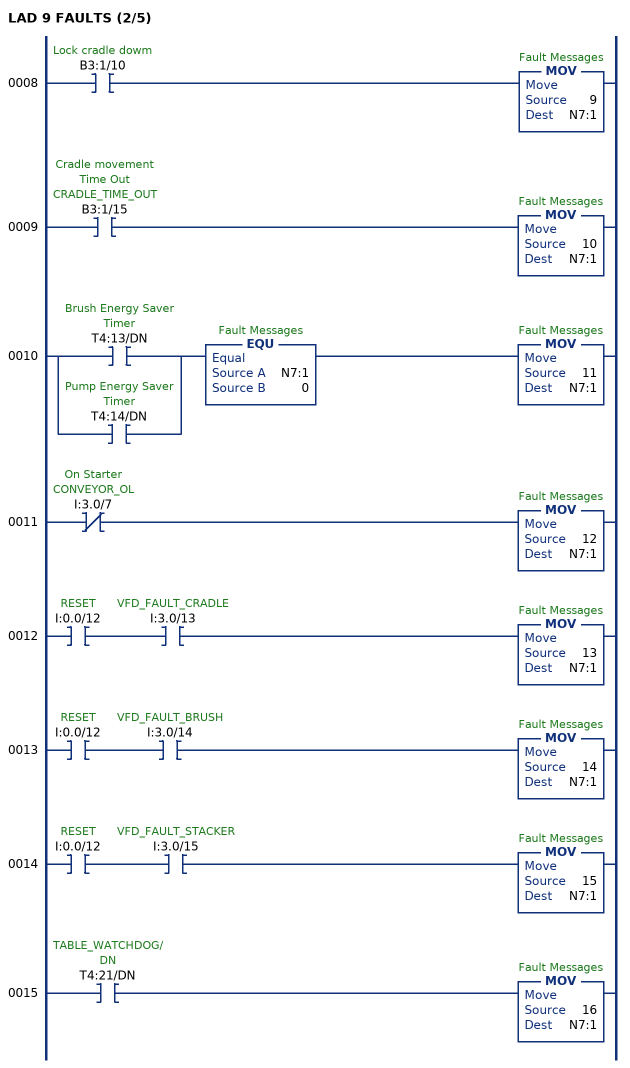
% Rung: 8 %
SOR XIC B3:1/10 MOV 9 N7:1 EOR
%   B3:1/10  "Lock cradle dowm" %
%   N7:1  "Fault Messages" %
% Rung: 9 %
SOR XIC B3:1/15 MOV 10 N7:1 EOR
%   B3:1/15  CRADLE_TIME_OUT  "Cradle movement Time Out" %
%   N7:1  "Fault Messages" %
% Rung: 10 %
SOR BST XIC T4:13/DN NXB XIC T4:14/DN BND EQU N7:1 0 MOV 11 N7:1 EOR
%   T4:13  "Brush Energy Saver Timer" %
%   T4:14  "Pump Energy Saver Timer" %
%   N7:1  "Fault Messages" %
% Rung: 11 %
SOR XIO I:3.0/7 MOV 12 N7:1 EOR
%   I:3.0/7  CONVEYOR_OL  "On Starter" %
%   N7:1  "Fault Messages" %
% Rung: 12 %
SOR XIC I:0.0/12 XIC I:3.0/13 MOV 13 N7:1 EOR
%   I:0.0/12  RESET %
%   I:3.0/13  VFD_FAULT_CRADLE %
%   N7:1  "Fault Messages" %
% Rung: 13 %
SOR XIC I:0.0/12 XIC I:3.0/14 MOV 14 N7:1 EOR
%   I:0.0/12  RESET %
%   I:3.0/14  VFD_FAULT_BRUSH %
%   N7:1  "Fault Messages" %
% Rung: 14 %
SOR XIC I:0.0/12 XIC I:3.0/15 MOV 15 N7:1 EOR
%   I:0.0/12  RESET %
%   I:3.0/15  VFD_FAULT_STACKER %
%   N7:1  "Fault Messages" %
% Rung: 15 %
SOR XIC T4:21/DN MOV 16 N7:1 EOR
%   T4:21  TABLE_WATCHDOG %
%   N7:1  "Fault Messages" %

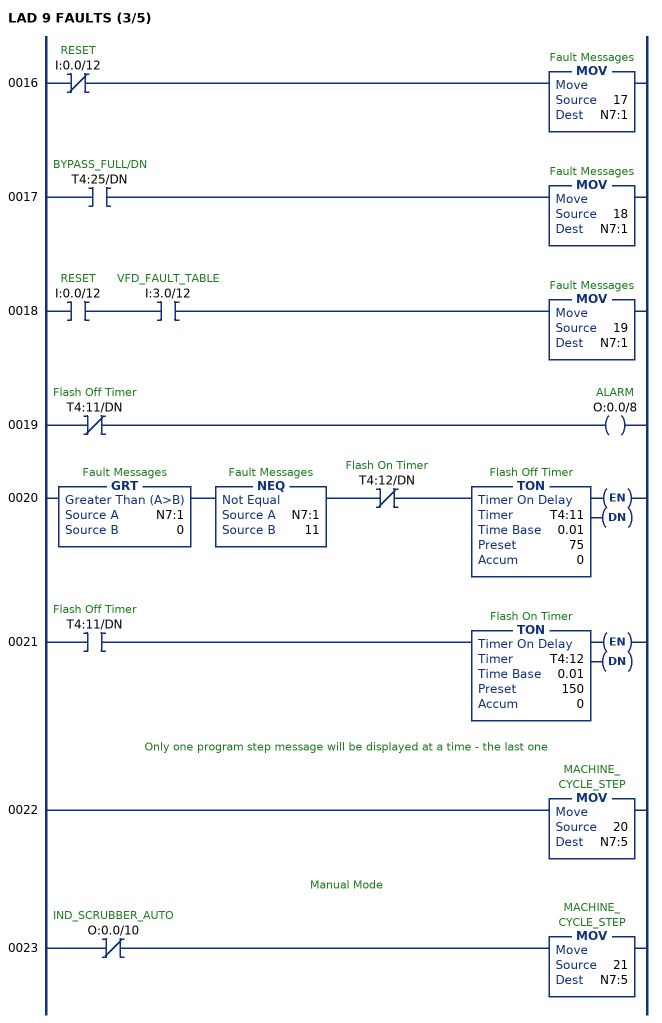
% Rung: 16 %
SOR XIO I:0.0/12 MOV 17 N7:1 EOR
%   I:0.0/12  RESET %
%   N7:1  "Fault Messages" %
% Rung: 17 %
SOR XIC T4:25/DN MOV 18 N7:1 EOR
%   T4:25  BYPASS_FULL %
%   N7:1  "Fault Messages" %
% Rung: 18 %
SOR XIC I:0.0/12 XIC I:3.0/12 MOV 19 N7:1 EOR
%   I:0.0/12  RESET %
%   I:3.0/12  VFD_FAULT_TABLE %
%   N7:1  "Fault Messages" %
% Rung: 19 %
SOR XIO T4:11/DN OTE O:0.0/8 EOR
%   T4:11  "Flash Off Timer" %
%   O:0.0/8  ALARM %
% Rung: 20 %
SOR GRT N7:1 0 NEQ N7:1 11 XIO T4:12/DN TON T4:11 0.01 75 0 EOR
%   N7:1  "Fault Messages" %
%   T4:12  "Flash On Timer" %
%   T4:11  "Flash Off Timer" %
% Rung: 21 %
SOR XIC T4:11/DN TON T4:12 0.01 150 0 EOR
%   T4:11  "Flash Off Timer" %
%   T4:12  "Flash On Timer" %
% Rung: 22 %
% Only one program step message will be displayed at a time - the last one %
SOR MOV 20 N7:5 EOR
%   N7:5  MACHINE_CYCLE_STEP %
% Rung: 23 %
% Manual Mode %
SOR XIO O:0.0/10 MOV 21 N7:5 EOR
%   O:0.0/10  IND_SCRUBBER_AUTO %
%   N7:5  MACHINE_CYCLE_STEP %

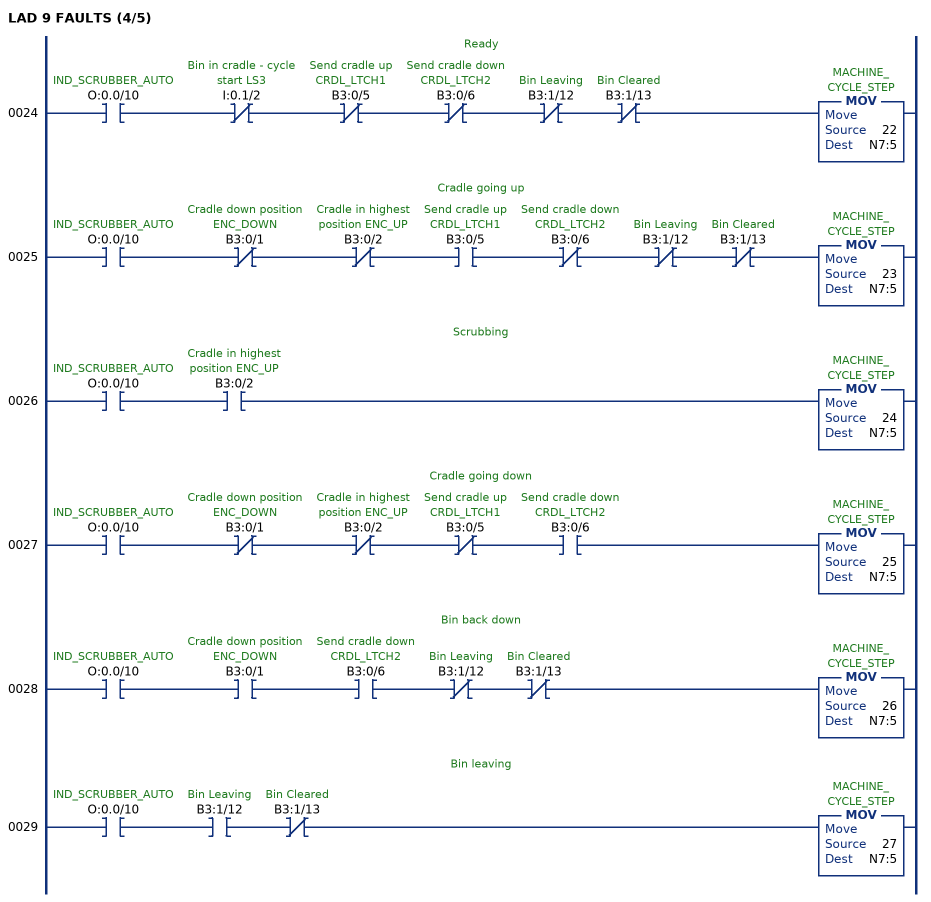
% Rung: 24 %
% Ready %
SOR XIC O:0.0/10 XIO I:0.1/2 XIO B3:0/5 XIO B3:0/6 XIO B3:1/12 XIO B3:1/13 MOV 22 N7:5 EOR
%   O:0.0/10  IND_SCRUBBER_AUTO %
%   I:0.1/2  LS3  "Bin in cradle - cycle start" %
%   B3:0/5  CRDL_LTCH1  "Send cradle up" %
%   B3:0/6  CRDL_LTCH2  "Send cradle down" %
%   B3:1/12  "Bin Leaving" %
%   B3:1/13  "Bin Cleared" %
%   N7:5  MACHINE_CYCLE_STEP %
% Rung: 25 %
% Cradle going up %
SOR XIC O:0.0/10 XIO B3:0/1 XIO B3:0/2 XIC B3:0/5 XIO B3:0/6 XIO B3:1/12 XIO B3:1/13 MOV 23 N7:5 EOR
%   O:0.0/10  IND_SCRUBBER_AUTO %
%   B3:0/1  ENC_DOWN  "Cradle down position" %
%   B3:0/2  ENC_UP  "Cradle in highest position" %
%   B3:0/5  CRDL_LTCH1  "Send cradle up" %
%   B3:0/6  CRDL_LTCH2  "Send cradle down" %
%   B3:1/12  "Bin Leaving" %
%   B3:1/13  "Bin Cleared" %
%   N7:5  MACHINE_CYCLE_STEP %
% Rung: 26 %
% Scrubbing %
SOR XIC O:0.0/10 XIC B3:0/2 MOV 24 N7:5 EOR
%   O:0.0/10  IND_SCRUBBER_AUTO %
%   B3:0/2  ENC_UP  "Cradle in highest position" %
%   N7:5  MACHINE_CYCLE_STEP %
% Rung: 27 %
% Cradle going down %
SOR XIC O:0.0/10 XIO B3:0/1 XIO B3:0/2 XIO B3:0/5 XIC B3:0/6 MOV 25 N7:5 EOR
%   O:0.0/10  IND_SCRUBBER_AUTO %
%   B3:0/1  ENC_DOWN  "Cradle down position" %
%   B3:0/2  ENC_UP  "Cradle in highest position" %
%   B3:0/5  CRDL_LTCH1  "Send cradle up" %
%   B3:0/6  CRDL_LTCH2  "Send cradle down" %
%   N7:5  MACHINE_CYCLE_STEP %
% Rung: 28 %
% Bin back down %
SOR XIC O:0.0/10 XIC B3:0/1 XIC B3:0/6 XIO B3:1/12 XIO B3:1/13 MOV 26 N7:5 EOR
%   O:0.0/10  IND_SCRUBBER_AUTO %
%   B3:0/1  ENC_DOWN  "Cradle down position" %
%   B3:0/6  CRDL_LTCH2  "Send cradle down" %
%   B3:1/12  "Bin Leaving" %
%   B3:1/13  "Bin Cleared" %
%   N7:5  MACHINE_CYCLE_STEP %
% Rung: 29 %
% Bin leaving %
SOR XIC O:0.0/10 XIC B3:1/12 XIO B3:1/13 MOV 27 N7:5 EOR
%   O:0.0/10  IND_SCRUBBER_AUTO %
%   B3:1/12  "Bin Leaving" %
%   B3:1/13  "Bin Cleared" %
%   N7:5  MACHINE_CYCLE_STEP %

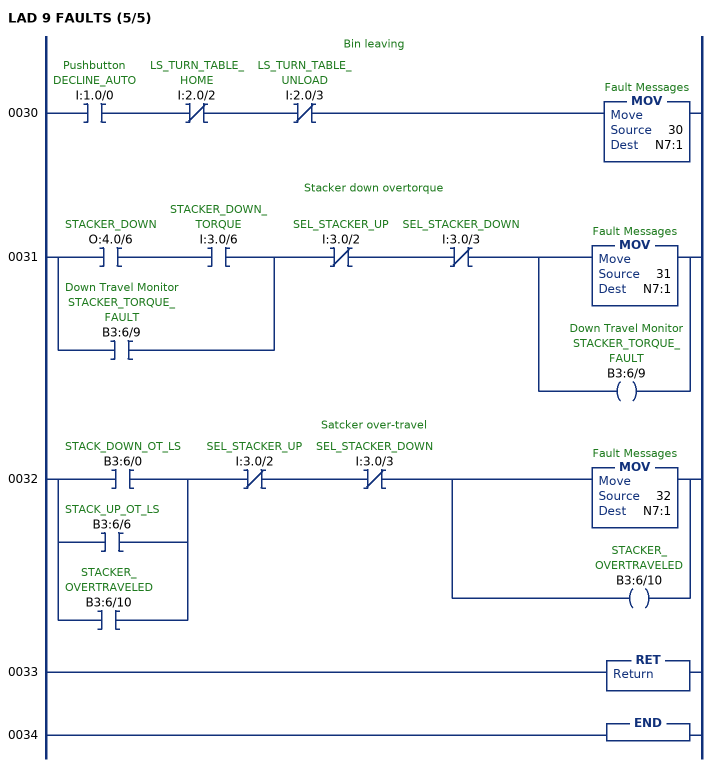
% Rung: 30 %
% Bin leaving %
SOR XIC I:1.0/0 XIO I:2.0/2 XIO I:2.0/3 MOV 30 N7:1 EOR
%   I:1.0/0  DECLINE_AUTO  "Pushbutton" %
%   I:2.0/2  LS_TURN_TABLE_HOME %
%   I:2.0/3  LS_TURN_TABLE_UNLOAD %
%   N7:1  "Fault Messages" %
% Rung: 31 %
% Stacker down overtorque %
SOR BST XIC O:4.0/6 XIC I:3.0/6 NXB XIC B3:6/9 BND XIO I:3.0/2 XIO I:3.0/3 BST MOV 31 N7:1 NXB OTE B3:6/9 BND EOR
%   O:4.0/6  STACKER_DOWN %
%   I:3.0/6  STACKER_DOWN_TORQUE %
%   B3:6/9  STACKER_TORQUE_FAULT  "Down Travel Monitor" %
%   I:3.0/2  SEL_STACKER_UP %
%   I:3.0/3  SEL_STACKER_DOWN %
%   N7:1  "Fault Messages" %
% Rung: 32 %
% Satcker over-travel %
SOR BST BST XIC B3:6/0 NXB XIC B3:6/6 BND NXB XIC B3:6/10 BND XIO I:3.0/2 XIO I:3.0/3 BST MOV 32 N7:1 NXB OTE B3:6/10 BND EOR
%   B3:6/0  STACK_DOWN_OT_LS %
%   B3:6/6  STACK_UP_OT_LS %
%   B3:6/10  STACKER_OVERTRAVELED %
%   I:3.0/2  SEL_STACKER_UP %
%   I:3.0/3  SEL_STACKER_DOWN %
%   N7:1  "Fault Messages" %
% Rung: 33 %
SOR RET EOR
% Rung: 34 %
SOR END EOR

LADDER 10 "SPARE"
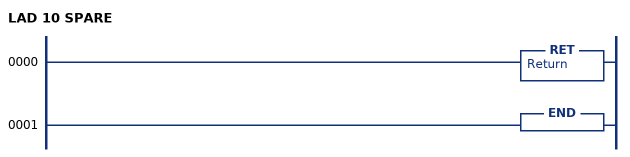
% Rung: 0 %
SOR RET EOR
% Rung: 1 %
SOR END EOR

LADDER 11 "DECLINE"
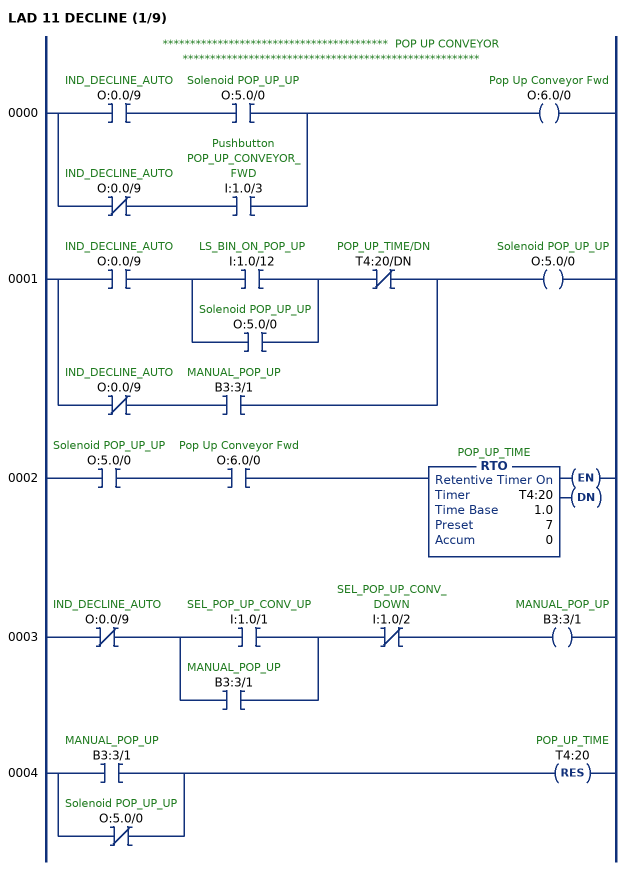
% Rung: 0 %
% *****************************************  POP UP CONVEYOR ****************************************************** %
SOR BST XIC O:0.0/9 XIC O:5.0/0 NXB XIO O:0.0/9 XIC I:1.0/3 BND OTE O:6.0/0 EOR
%   O:0.0/9  IND_DECLINE_AUTO %
%   O:5.0/0  POP_UP_UP  "Solenoid" %
%   I:1.0/3  POP_UP_CONVEYOR_FWD  "Pushbutton" %
%   O:6.0/0  "Pop Up Conveyor Fwd" %
% Rung: 1 %
SOR BST XIC O:0.0/9 BST XIC I:1.0/12 NXB XIC O:5.0/0 BND XIO T4:20/DN NXB XIO O:0.0/9 XIC B3:3/1 BND OTE O:5.0/0 EOR
%   O:0.0/9  IND_DECLINE_AUTO %
%   I:1.0/12  LS_BIN_ON_POP_UP %
%   O:5.0/0  POP_UP_UP  "Solenoid" %
%   T4:20  POP_UP_TIME %
%   B3:3/1  MANUAL_POP_UP %
% Rung: 2 %
SOR XIC O:5.0/0 XIC O:6.0/0 RTO T4:20 1.0 7 0 EOR
%   O:5.0/0  POP_UP_UP  "Solenoid" %
%   O:6.0/0  "Pop Up Conveyor Fwd" %
%   T4:20  POP_UP_TIME %
% Rung: 3 %
SOR XIO O:0.0/9 BST XIC I:1.0/1 NXB XIC B3:3/1 BND XIO I:1.0/2 OTE B3:3/1 EOR
%   O:0.0/9  IND_DECLINE_AUTO %
%   I:1.0/1  SEL_POP_UP_CONV_UP %
%   B3:3/1  MANUAL_POP_UP %
%   I:1.0/2  SEL_POP_UP_CONV_DOWN %
% Rung: 4 %
SOR BST XIC B3:3/1 NXB XIO O:5.0/0 BND RES T4:20 EOR
%   B3:3/1  MANUAL_POP_UP %
%   O:5.0/0  POP_UP_UP  "Solenoid" %
%   T4:20  POP_UP_TIME %

